TYPE ST_DoDi_out :
STRUCT
	DO0	AT %Q*	: BOOL;
END_STRUCT
END_TYPE

(* stored: Version 1.1.0.1, ProductVersion 3.1.4024.9
   DUT ST_DoDi_out: Id {89c07b4a-9298-45c6-b5f6-8ce2a842324a} *)
